// Mitsubishi GX Works2 project: 240430_timechart09_음변환   PLC: Q03UDV

PROGRAM MAIN
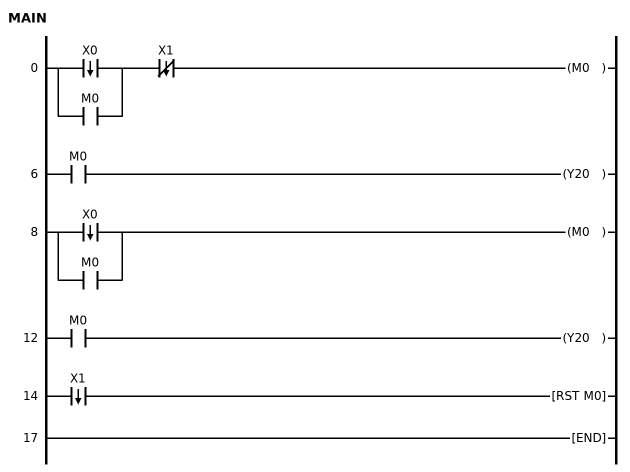
0     LDF     X0
      OR      M0
      ANDFI   X1
      OUT     M0
6     LD      M0
      OUT     Y20
8     LDF     X0
      OR      M0
      OUT     M0
12    LD      M0
      OUT     Y20
14    LDF     X1
      RST     M0
17    END
END_PROGRAM
